(* PLC project 07_r_trig.project, CODESYS CODESYS V3.5 SP22 Patch 2 *)
(* stored: creationDateTime 2026-07-24T05:19:27.9688479, modificationDateTime 2026-07-24T05:19:16.4040579 *)

PROGRAM PLC_PRG
  VAR
    fbRise : Standard.R_TRIG;
    xInput : BOOL;
    xPulse : BOOL;
    xExecuted : BOOL;
  END_VAR

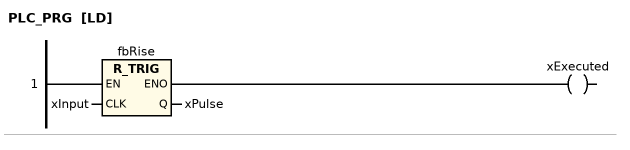
(* LD diagram, written out as Structured Text *)

fbRise(CLK := xInput, Q => xPulse);
xExecuted := fbRise.ENO;
END_PROGRAM

CONFIGURATION Application
  RESOURCE Application ON PLC
    TASK MainTask(INTERVAL := T#20ms, PRIORITY := 1);
    PROGRAM PLC_PRG WITH MainTask : PLC_PRG;
  END_RESOURCE
END_CONFIGURATION
